(* PLC project Senza_nome, Sconosciuto Senza_nome 1 *)
(* stored: creationDateTime 2026-09-02T10:36:19, modificationDateTime 2026-09-02T11:05:24 *)

PROGRAM program0
  VAR
    STOP : BOOL;
    S1 : BOOL;
    S2 : BOOL;
    LAMPADA_MARCIA_AVANTI : BOOL;
    LAMPADA_MARCIA_INDIETRO : BOOL;
    LAMPADA_SEGNALAZIONE_FUNZIONAMENTO : BOOL;
    M1 : BOOL;
    M2 : BOOL;
  END_VAR

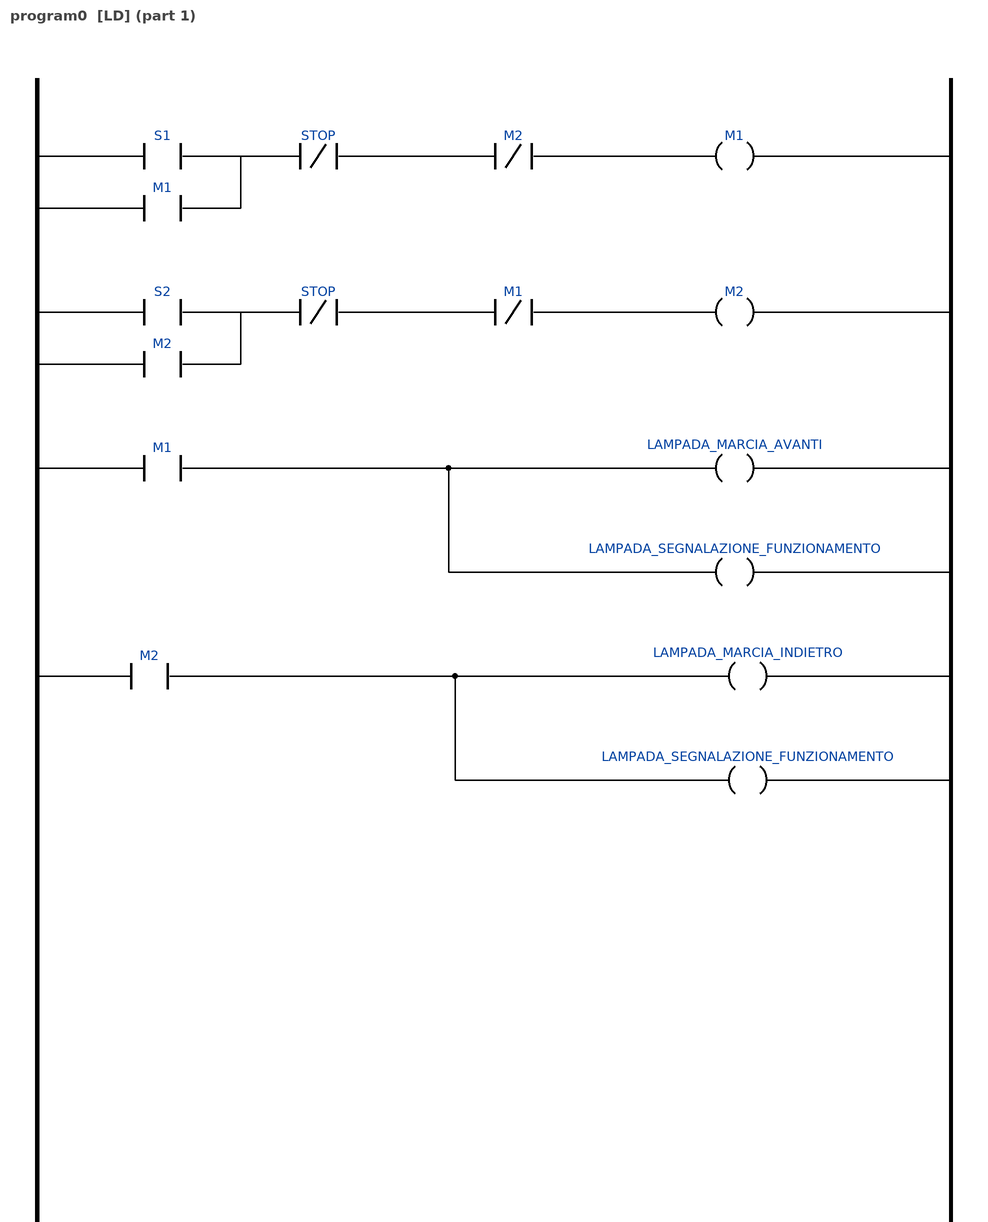
(* LD diagram, written out as Structured Text *)
M1 := (S1 OR M1) AND NOT STOP AND NOT M2;
M2 := (S2 OR M2) AND NOT STOP AND NOT M1;
LAMPADA_MARCIA_AVANTI := M1;
LAMPADA_MARCIA_INDIETRO := M2;
LAMPADA_SEGNALAZIONE_FUNZIONAMENTO := M1;
LAMPADA_SEGNALAZIONE_FUNZIONAMENTO := M2;
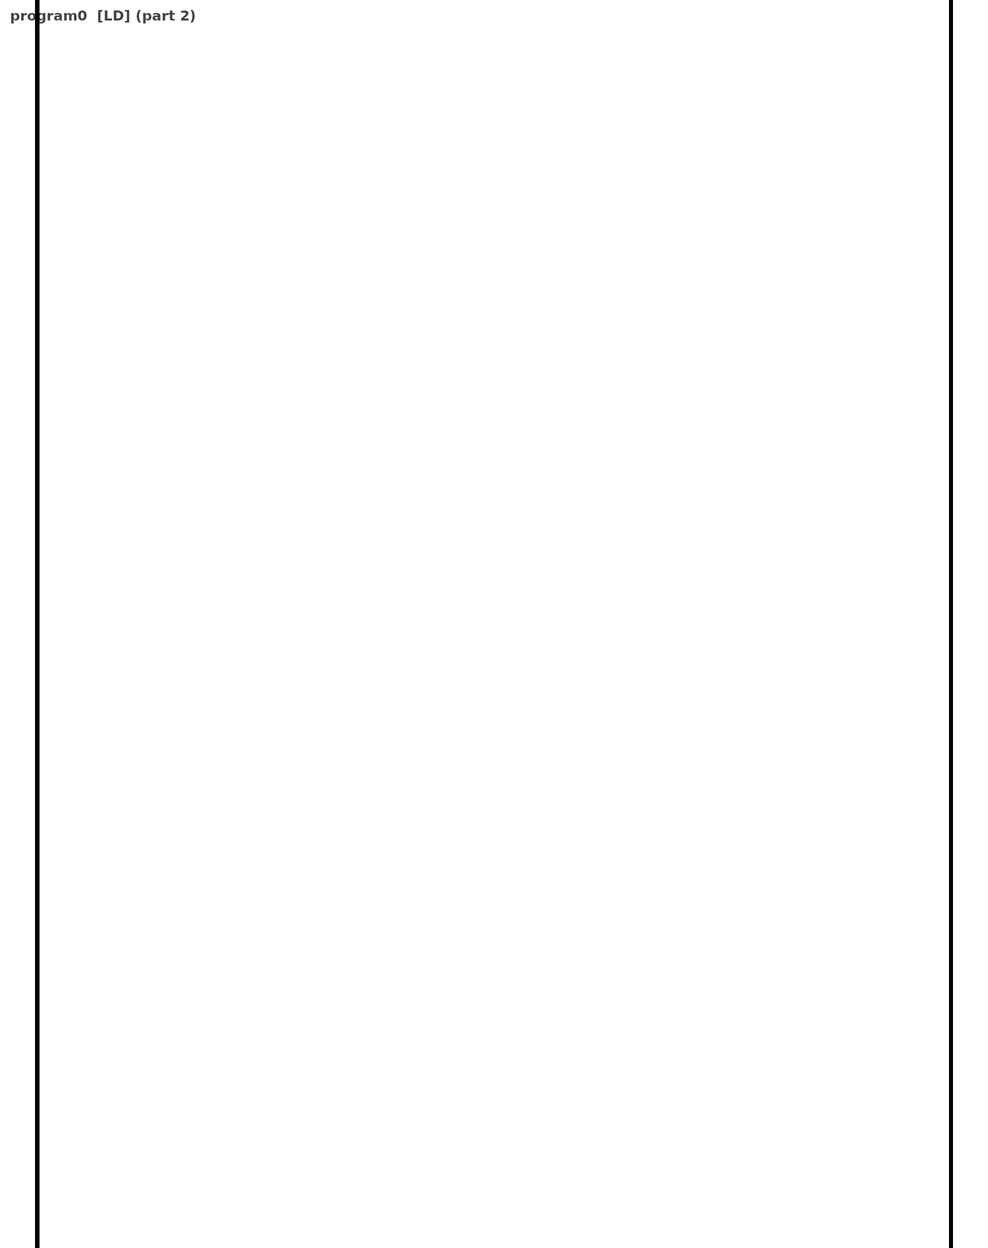
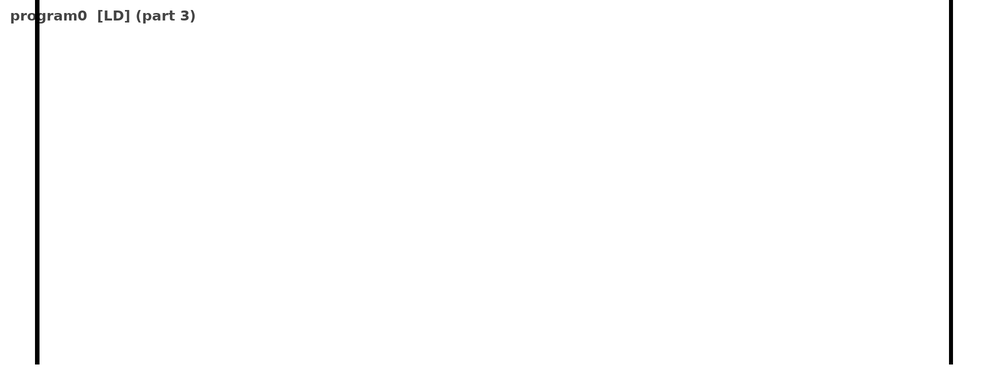
END_PROGRAM

CONFIGURATION Config0
  RESOURCE Res0 ON PLC
    TASK task0(INTERVAL := T#20ms, PRIORITY := 0);
    PROGRAM instance0 WITH task0 : program0;
  END_RESOURCE
END_CONFIGURATION
